Fanuc TP program (LS listing): HF_VAC_ON.LS

/PROG  HF_VAC_ON
/ATTR
OWNER		= MNEDITOR;
COMMENT		= "Vacuum On";
PROG_SIZE	= 620;
CREATE		= DATE 20-06-29  TIME 11:06:30;
MODIFIED	= DATE 21-05-13  TIME 13:54:42;
FILE_NAME	= T_VACON;
VERSION		= 0;
LINE_COUNT	= 25;
MEMORY_SIZE	= 1064;
PROTECT		= READ_WRITE;
TCD:  STACK_SIZE	= 0,
      TASK_PRIORITY	= 50,
      TIME_SLICE	= 0,
      BUSY_LAMP_OFF	= 0,
      ABORT_REQUEST	= 0,
      PAUSE_REQUEST	= 0;
DEFAULT_GROUP	= *,*,*,*,*;
CONTROL_CODE	= 00000000 00000000;
/APPL
/MN
   1:  --eg:Vacuum On
    :  --kn:KANJI Vacuum On
    :  --ch:Vacuum On ;
   2:  $WAITTMOUT=500 ;
   3:   ;
   4:  RO[1:VACUUM]=OFF ;
   5:  WAIT    .50(sec) ;
   6:  WAIT RI[1:Vacuum Switch Sensor]=ON TIMEOUT,LBL[9114] ;
   7:  WAIT RI[3:Cylinder RTR]=ON TIMEOUT,LBL[9111] ;
   8:  JMP LBL[9999] ;
   9:   ;
  10:   ;
  11:   ;
  12:  !Cylinder Extension Timeout ;
  13:  LBL[9111:Error] ;
  14:  R[240:ERROR_STATE]=111    ;
  15:  JMP LBL[9000] ;
  16:   ;
  17:  !Vacuum Pressure Low Timeout ;
  18:  LBL[9114] ;
  19:  R[240:ERROR_STATE]=114    ;
  20:  JMP LBL[9000] ;
  21:   ;
  22:  LBL[9000:Error] ;
  23:  CALL HF_ERRORLOOP    ;
  24:   ;
  25:  LBL[9999:End] ;
/POS
/END
